(* CODESYS project OwenModules.export

Project tree, tasks and I/O mapping:
  Owen/
    data type MV210_101
    data type MV210_102
    data type MV210_212
    data type MV210_403
    data type PLC210_11
    data type _LeftSide
    data type _RightSide
*)

// Owen/MV210_101
TYPE MV210_101 :
STRUCT
	Exclude	:	BIT;
	Error	:	BIT;
	WriteSettings	:	BIT;
	ReadSettings	:	BIT;
	NewSettings	:	ARRAY [1..8] OF ANALOG_SENSOR_SETTINGS;
	OldSettings	:	ARRAY [1..8] OF ANALOG_SENSOR_SETTINGS;
	Ch	:	ARRAY [1..8] OF ANALOG_SENSOR_VALUE;
END_STRUCT
END_TYPE

// Owen/MV210_102
TYPE MV210_102 :
STRUCT
	Exclude	:	BIT;
	Error	:	BIT;
	WriteSettings	:	BIT;
	ReadSettings	:	BIT;
	NewSettings	:	ARRAY [1..8] OF FAST_ANALOG_SENSOR_SETTINGS;
	OldSettings	:	ARRAY [1..8] OF FAST_ANALOG_SENSOR_SETTINGS;
	Ch	:	ARRAY [1..8] OF ANALOG_SENSOR_VALUE;
END_STRUCT
END_TYPE

// Owen/MV210_212
TYPE MV210_212 :
STRUCT
	Exclude	:	BIT;
	Error	:	BIT;
	Ch		:	DWORD;
END_STRUCT
END_TYPE

// Owen/MV210_403
TYPE MV210_403 :
STRUCT
	Exclude	:	BIT;
	Error	:	BIT;
	ChRead	:	DWORD;
	Ch		:	DWORD;
END_STRUCT
END_TYPE

// Owen/PLC210_11
TYPE PLC210_11 :
STRUCT
	LeftSide	:	_LeftSide;
	RightSide	:	_RightSide;
END_STRUCT
END_TYPE

// Owen/_LeftSide
TYPE _LeftSide :
STRUCT
	DiCh	:	DWORD;
	DoCh	:	DWORD;
END_STRUCT
END_TYPE

// Owen/_RightSide
TYPE _RightSide :
STRUCT
	DoCh	:	DWORD;
END_STRUCT
END_TYPE
